Universal Robots PolyScope program: move_path_1.urp

Program move_path_1 (installation=default directory=/programs createdIn=5.14.5 lastSavedIn=5.14.5 robotSerialNumber=20236801216)
Calibrated DH parameters: a=[-0.000021, -0.748897, -0.28186, -0.00004, -0.000055, 0]; d=[0.236225, -424.082933, -1564.66872, 1988.95162, 0.159094, 0.153873]; alpha=[1.570844, 0.001002, 0.000337, 1.571488, -1.569996, 0]; deltaTheta=[0, -0.516316, 5.626292, 1.173211, 0.000001, 0]
InitVariablesNode
Robot Program (runOnlyOnce=false)
  pa1 := path1[1]
  pa2 := path1[2]
  p1 := path1[3]
  p2 := path1[4]
  p3 := path1[5]
  p4 := path1[6]
  p5 := path1[7]
  pr1 := path1[8]
  Popup Message (haltProgram=false inputType=Variable) variable=pa1
  Popup Message (haltProgram=false inputType=Variable) variable=pa2
  Popup Message (haltProgram=false inputType=Variable) variable=p1
  Popup Message (haltProgram=false inputType=Variable) variable=p2
  Popup Message (haltProgram=false inputType=Variable) variable=p3
  Popup Message (haltProgram=false inputType=Variable) variable=p4
  Popup Message (haltProgram=false inputType=Variable) variable=p5
  Popup Message (haltProgram=false inputType=Variable) variable=pr1
  MoveJ speed 60 deg/s, acceleration 80 deg/s^2 (useActiveTCP=true) feature=Base
    Waypoint Waypoint_1: TCP in base x=-372.861 y=716.17 z=314.677 mm, rx=1.5708 ry=0 rz=0 rad; joints [-79.161, -60.426, 105.047, -44.564, -79.226, 359.93] deg; TCP offset x=0 y=0 z=19 mm, rx=0 ry=0 rz=0 rad
  MoveJ speed 60 deg/s, acceleration 80 deg/s^2 (useActiveTCP=true) feature=Base
    Waypoint Variable (Variable): variable=pa1
  MoveL speed 200 mm/s, acceleration 1200 mm/s^2 (useActiveTCP=true) feature=Base
    Waypoint Variable (Variable): variable=pa2
  MoveL speed 50 mm/s, acceleration 1200 mm/s^2 (useActiveTCP=true) feature=Base
    Waypoint Variable (Variable): variable=p1
  Wait Sleep waitTime=1
  MoveP speed 12 mm/s, acceleration 1200 mm/s^2 (blendRadius=0.025 useActiveTCP=true) feature=Base
    Waypoint Variable (Variable): variable=p2
  MoveP speed 6 mm/s, acceleration 1200 mm/s^2 (blendRadius=0.025 useActiveTCP=true) feature=Base
    CircleMove (OrientationMode=FIXED)
      Waypoint Variable (Variable): variable=p3
      Waypoint Variable (Variable): variable=p4
  MoveP speed 12 mm/s, acceleration 1200 mm/s^2 (blendRadius=0.025 useActiveTCP=true) feature=Base
    Waypoint Variable (Variable): variable=p5
  MoveL speed 250 mm/s, acceleration 1200 mm/s^2 (useActiveTCP=true) feature=Base
    Waypoint Variable (Variable): variable=pr1
  MoveJ speed 60 deg/s, acceleration 80 deg/s^2 (useActiveTCP=true) feature=Base
    Waypoint Waypoint_1: TCP in base x=-372.861 y=716.17 z=314.677 mm, rx=1.5708 ry=0 rz=0 rad; joints [-79.161, -60.426, 105.047, -44.564, -79.226, 359.93] deg
